PROGRAM MAIN
VAR
	
 
END_VAR

A_1_PRG_Main_Master();

END_PROGRAM

(* stored: Version 1.1.0.1, ProductVersion 3.1.4026.17
   POU MAIN: Id {278d4c6c-3780-4c87-a241-22c3aeef8360}, SpecialFunc None *)
